INTERFACE I_Drive

{attribute 'monitoring':='call'}
PROPERTY Active : BOOL
GET
END_GET
END_PROPERTY

{attribute 'monitoring':='call'}
PROPERTY AtHome : BOOL
GET
END_GET
END_PROPERTY

{attribute 'monitoring':='call'}
PROPERTY Error : BOOL
GET
END_GET
END_PROPERTY

{attribute 'monitoring':='call'}
PROPERTY HomeSet : BOOL
GET
END_GET
END_PROPERTY

METHOD ABSTRACT homingSequence : BOOL
VAR_INPUT
END_VAR
END_METHOD

METHOD reset : BOOL
VAR_INPUT
END_VAR
END_METHOD

METHOD ABSTRACT stop : BOOL
VAR_INPUT
END_VAR
END_METHOD

METHOD toHome : BOOL
VAR_INPUT
END_VAR
END_METHOD

END_INTERFACE

(* stored: Version 1.1.0.1, ProductVersion 3.1.4024.11
   Itf I_Drive: Id {aada4de7-926f-4d11-a81f-b2f83520ca8a}
   Property Active: Id {9a2d2db7-998b-4a1e-951d-f922ab09002a}
   Get Get: Id {6915a7a6-80a8-4e99-9766-da284d366648}
   Property AtHome: Id {c945b7b3-2b07-4ade-bec7-db86b1867d6e}
   Get Get: Id {0916b128-855e-4c40-abca-18ae2e234caf}
   Property Error: Id {d763e159-5055-4093-ba37-2326046f7fb3}
   Get Get: Id {331ed520-01e3-49cd-9125-89f5ecb7e543}
   Property HomeSet: Id {59aa46b5-e497-4d28-b1ac-2fb03365670d}
   Get Get: Id {8d08c66a-11a3-42d2-9608-164b61089ebd}
   Method homingSequence: Id {373dfb60-8328-4625-88c4-989f0120ef66}
   Method reset: Id {0d9d3e3a-bbdd-4587-93f0-d6e87f5df259}
   Method stop: Id {b9c17277-e722-484b-ad84-dc2b3100a9ef}
   Method toHome: Id {ce068013-3c22-478e-8dc0-fe2b808f5b6c} *)
